FUNCTION_BLOCK Controler
  (* Standard: 61499-2 *)
  (* Version 0,1, 2015-00-07, Th?o, PC_THEO *)
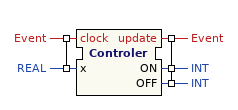
  EVENT_INPUT
    clock WITH x;
  END_EVENT
  EVENT_OUTPUT
    update WITH ON, OFF;
  END_EVENT
  VAR_INPUT
    x : REAL;
  END_VAR
  VAR_OUTPUT
    ON : INT;
    OFF : INT;
  END_VAR
  VAR
    timer : BOOL;
  END_VAR
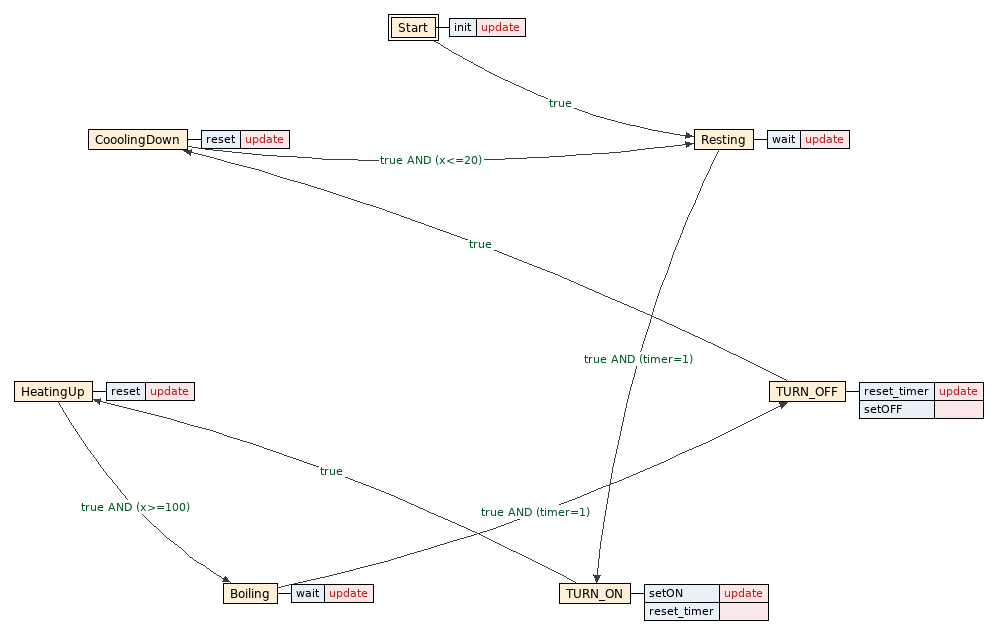
  EC_STATES
    Start : init -> update;
    Resting : wait -> update;
    TURN_OFF : reset_timer -> update, setOFF;
    TURN_ON : setON -> update, reset_timer;
    Boiling : wait -> update;
    HeatingUp : reset -> update;
    CooolingDown : reset -> update;
  END_STATES
  EC_TRANSITIONS
    Resting TO TURN_ON := true AND (timer=1);
    TURN_OFF TO CooolingDown := true;
    TURN_ON TO HeatingUp := true;
    Boiling TO TURN_OFF := true AND (timer=1);
    HeatingUp TO Boiling := true AND (x>=100);
    CooolingDown TO Resting := true AND (x<=20);
    Start TO Resting := true;
  END_TRANSITIONS
  ALGORITHM setON IN C:
me->ON=1;
printf("setON\n");
  END_ALGORITHM
  ALGORITHM setOFF IN C:
me->OFF=1;
printf("setOFF\n");
  END_ALGORITHM
  ALGORITHM wait IN C:
sleep(1);
me->timer=1;
  END_ALGORITHM
  ALGORITHM reset_timer IN C:
me->timer=0;
  END_ALGORITHM
  ALGORITHM reset IN C:
me->ON=0; me->OFF=0;
  END_ALGORITHM
  ALGORITHM init IN C:
me->ON=0; me->OFF=0;
me->timer=0;
me->x=20;
  END_ALGORITHM
END_FUNCTION_BLOCK
